PROGRAM MAIN
VAR
END_VAR

END_PROGRAM

(* stored: Version 1.1.0.1
   POU MAIN: Id {c425906c-7d9c-4c38-b135-c08afdf69580} *)
